Staubli VAL3: sendMoving.pgx

program sendMoving()
  local num buffer[4]
begin
  buffer[0] = MAGIC_HEADER
  buffer[1] = 132
  buffer[2] = sel(isSettled(), 1, 0)
  sioSet(socket, buffer)
end
